(* CODESYS project PID_regulator.project

Project tree, tasks and I/O mapping:
  Device : CODESYS Control Win V3, 3S - Smart Software Solutions GmbH, order no. 305021, version 3.5.4.10
    application Application
      libraries: Standard, * (System)
      task MainTask (cyclic, interval t#20ms, priority 1) calls PID_Tank
      global variables GVL_Input
      global variables GVL_Output
      global variables GVL_Memory
      global variables GVL_Data
      PID/
        function block PID_regulator [ST]
      Progs/
        program PID_Tank [LD]
      Models/
        function block Tank [ST]
        function block HeatExchanger2 [ST]
      Symbols
  text list GlobalTextList
*)

// Device/Application/GVL_Input
VAR_GLOBAL
	Knapp1: BOOL; // Knapp på våning 1
	Knapp2: BOOL; // 
	Knapp3: BOOL;
	Knapp4: BOOL;
	Vaning1 :BOOL;
	Vaning2 :BOOL;
	Vaning3 :BOOL;
	Vaning4 :BOOL;
	Manuell :BOOL;
	Auto :BOOL;
	Upp :BOOL;
	Ner  :BOOL;
	Service_reset :BOOL;
END_VAR

// Device/Application/GVL_Output
VAR_GLOBAL
	Lampa1 :BOOL;
	Lampa2 :BOOL;
	Lampa3 :BOOL;
	Lampa4 :BOOL;
	HissUpp :BOOL;
	HissNer :BOOL;
	HissDorr :BOOL;
	LampaAuto :BOOL;
	
END_VAR

// Device/Application/GVL_Memory
VAR_GLOBAL
END_VAR

// Device/Application/GVL_Data
VAR_GLOBAL
	PV_tank: REAL;
	SP_tank: REAL := 50.0;
	Kc_tank: REAL := 3.0;
	Ti_tank: REAL := 10.0;
	Td_tank: REAL := 0.0;
	Out_tank: REAL := 0.0;
	Inflode: REAL;
	Utflode: REAL := 50;
	PID_out: REAL;
	P_tank: REAL;
	I_tank: REAL;
	D_tank: REAL;
	Tank_niva: REAL;
	HMI_Start_Stopp: BOOL;
	HMI_Tank_Reset: BOOL;
	HMI_PID_Auto: BOOL;
	HMI_Out: REAL;
END_VAR

// Device/Application/Progs/PID_Tank
PROGRAM PID_Tank
VAR
	PID_1: PID_regulator;
	Coca_Cola_Tank: Tank;
END_VAR

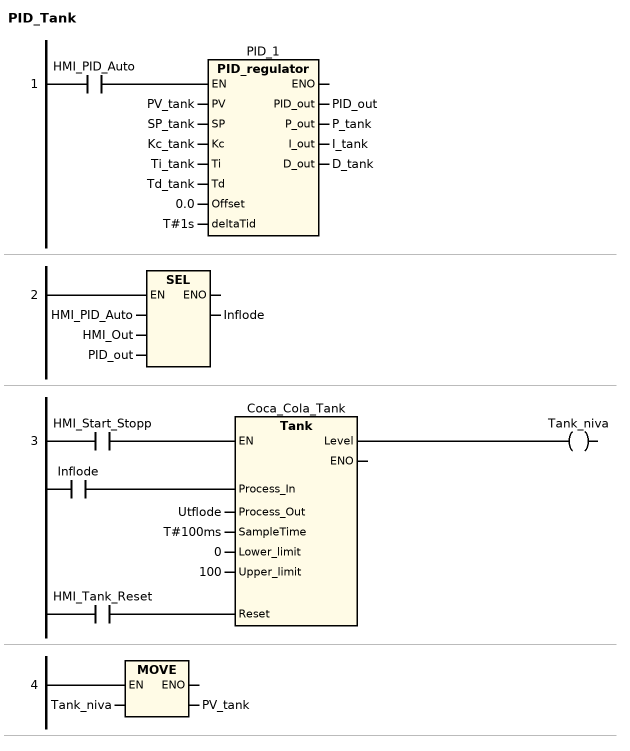
// NETWORK 1
PID_1(
    EN := HMI_PID_Auto,
    PV := PV_tank,
    SP := SP_tank,
    Kc := Kc_tank,
    Ti := Ti_tank,
    Td := Td_tank,
    Offset := 0.0,
    deltaTid := T#1s,
    PID_out => PID_out,
    P_out => P_tank,
    I_out => I_tank,
    D_out => D_tank); // PID_regulator

// NETWORK 2
Inflode := SEL(HMI_PID_Auto, HMI_Out, PID_out);

// NETWORK 3
Coca_Cola_Tank(
    EN := HMI_Start_Stopp,
    Process_In := Inflode,
    Process_Out := Utflode,
    SampleTime := T#100ms,
    Lower_limit := 0,
    Upper_limit := 100,
    Reset := HMI_Tank_Reset); // Tank
Tank_niva := Coca_Cola_Tank.Level;

// NETWORK 4
PV_tank := Tank_niva;

END_PROGRAM

// Device/Application/PID/PID_regulator
//***************************************************************
//* En enkel PID regulator för Codesys
//***************************************************************
FUNCTION_BLOCK PID_regulator
VAR_INPUT
	EN : BOOL;
	PV : REAL; //0-100%
	SP : REAL; //0-100%
	Kc : REAL;
	Ti : REAL; //i sekunder, 0=avstängd
	Td : REAL; //i sekunder
	Offset : REAL; //Offset för P om inte I används
	deltaTid: TIME; //Tid sedan senaste anrop
END_VAR
VAR_OUTPUT
	ENO : BOOL;
	PID_out: REAL; //Regulatorns utsignal
	P_out: REAL; //P-delens tillskott
	I_out: REAL; //I-delens tillskott
	D_out: REAL; //D-delens tillskott
END_VAR
VAR CONSTANT
	MILLIS: UINT := 1000;
	LOWERLIMIT: REAL := 0;
	UPPERLIMIT: REAL := 100;
END_VAR
VAR
	now: TIME := T#0S;
	lastTime: TIME := T#0S;
	err: REAL := 0; //Process error
	delta_t: REAL;
	lastPV: REAL := 0;
END_VAR

now := TIME();
IF EN = FALSE THEN
	ENO := FALSE;
ELSIF EN AND ((now - lastTime) > deltaTid) THEN
	err := SP - PV;
	delta_t := TIME_TO_REAL(deltaTid)/MILLIS;

	//Ti = 0, ingen integration, använd Offset
	IF Ti = 0 THEN
		P_out := Kc * err + Offset;
		I_out := 0;
	ELSE
		P_out := Kc * err;
		I_out := I_out + 1/Ti * P_out * delta_t;
	END_IF
	//wind-up för I_out
	IF I_out < LOWERLIMIT THEN
		I_out := LOWERLIMIT;
	ELSIF I_out > UPPERLIMIT THEN
		I_out := UPPERLIMIT;
	END_IF;
	
	//Observe that d(err)/dt = d(SP)/dt - d(PV)/dt
	//If SP constant,
	//d(err)/dt = - d(PV)/dt
	//Good: no output spikes
	//Bad: some processes need more aggressive tuning
	IF delta_t > 0 THEN
		D_out := Td * (PV - lastPV)/delta_t;
	END_IF;
	
	PID_out := P_out + I_out + D_out;
	//wind-up för PID_out
	IF PID_out < LOWERLIMIT THEN
		PID_out := LOWERLIMIT;
	ELSIF PID_out > UPPERLIMIT THEN
		PID_out := UPPERLIMIT;
	END_IF;
	
	lastTime := now;
	lastPV := PV;
	ENO := TRUE;
END_IF;

END_FUNCTION_BLOCK

// Device/Application/Models/Tank
//A.J. Jaworowski 2015-02-20
//Simulering av en tank med RedBull
FUNCTION_BLOCK Tank
VAR_INPUT
	EN: BOOL;
	Process_In: REAL;  //Flöde in per sekund, testa vad som händer on du matar in 100
					   //Därefter ska regulatorns OUT in i denna ingång.
	Process_Out: REAL; //Flöde ut per sekund, typ 90
					   //Effekten blir att tanken fylls med 10 per sekund
					   //Full efter ca 1 minut - testa
	SampleTime: TIME;  //Uppdateringstid, typ 100ms
	Lower_limit: REAL; //Tankens lägsta nivå, typ 0
	Upper_limit: REAL; //Tankens max nivå, kanske 500
	Reset: BOOL;
END_VAR
VAR_OUTPUT
	ENO: BOOL;
	Level: REAL; //Nivån i tanken
END_VAR
VAR
	now: TIME;
	lastTime: TIME;
	proc_sum_in: REAL := 0;
	proc_sum_out: REAL := 0;
	temp: REAL;
	millis: UINT := 1000;
	proc_out: REAL;
END_VAR

now := TIME();
IF Reset THEN
	Level := 0;
	lastTime := T#0S;
ELSIF EN THEN
	IF ((now - lastTime) > SampleTime) THEN
		Level := Level +  TIME_TO_REAL(SampleTime)/millis * (Process_In - Process_Out);
		IF Level < Lower_limit THEN
			Level := Lower_limit;
		ELSIF Level > Upper_limit THEN
			Level := Upper_limit;
		END_IF;
		lastTime := now;
		ENO := TRUE;
	END_IF;
END_IF;

END_FUNCTION_BLOCK

// Device/Application/Models/HeatExchanger2
// AJ Jaworowski 2015-02-23
// Following the presentation on
// http://openenergymonitor.org/emon/node/2999
FUNCTION_BLOCK HeatExchanger2
VAR_INPUT
	Heat_In:		REAL;		//In principle a radiator in the room [W]
	U:				REAL;		//Thermal conductance [W/K]
	TC:				REAL;		//Thermal capacity [J/K], commonly cv, specific heat capacity [J/kgK]
								//we use a smaller value than in reality, so that we can see changes
								//during a life-time...
	Temp_In:		REAL;		//Start temperature in the room [K]
	Temp_Out:		REAL;		//Outside temperature [K] 
	Sample_time:	TIME;
END_VAR
VAR_OUTPUT
	Temp:			REAL;		//The resulting room temperature
END_VAR
VAR
	now: TIME;
	lastTime: TIME := T#0s;
	delta_t: REAL;
	heat_flow: REAL;
	lastTemp: REAL;
END_VAR
VAR CONSTANT
	millis: REAL := 1000;
END_VAR

now := TIME();
IF ((now - lastTime) > Sample_time) THEN
	delta_t := TIME_TO_REAL(Sample_time)/millis;
	
	//First calculate net heat
	//Heat_In is our heat source
	//Second term is heat flow depending on temperature difference
	//Obs: At start, set lastTime to start temp Temp_In
	IF lastTime = T#0S THEN
		lastTemp := Temp_In;
	END_IF
	heat_flow := Heat_In - U * (lastTemp - Temp_Out);
	
	//Second: calculate temperature change due to heat_flow
	Temp := lastTemp + heat_flow * delta_t / TC;
	
	//Update variables for next iteration
	lastTemp := Temp;
	lastTime := now;
END_IF;

END_FUNCTION_BLOCK
